# EPICS autosave request: iocBoot/gmca_23o_ioc1/dbSave/HD_St_.req
%
% BURT Request File
%
% $(P)HD:St:  Horiz Deflecting mirror Z-positioning
%

file assy.req ASSY=$(P)HD:St
$(P)HD:St:Base1:23
$(P)HD:St:Base23
file mtr1.req MTR1=$(P)HD:mz1
file mtr1.req MTR1=$(P)HD:mz2
file mtr1.req MTR1=$(P)HD:mz3
file drv1.req DRV1=$(P)HD:SZ1
file drv1.req DRV1=$(P)HD:SZ2
file drv1.req DRV1=$(P)HD:SZ3
file axs1.req AXS1=$(P)HD:SL
file axs1.req AXS1=$(P)HD:HT
file axs1.req AXS1=$(P)HD:HR
